// Mitsubishi GX Works2 project: 타이머1   PLC: Q02/Q02H

PROGRAM MAIN
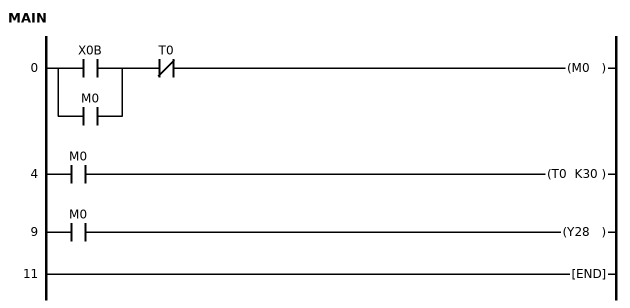
0     LD      X0B
      OR      M0
      ANI     T0
      OUT     M0
4     LD      M0
      OUT     T0 K30
9     LD      M0
      OUT     Y28
11    END
END_PROGRAM
